// TwinCAT 3 PLC project plc_tmo_granite3_test
// ProgramVersion: 3.1.4022.7
// libraries:
//   LCLS General, * (SLAC)
//   lcls-twincat-motion, * (SLAC)
//   lcls2-cc-lib, * (SLAC)
//   PMPS, * (SLAC - LCLS)
//   Tc2_Standard, * (Beckhoff Automation GmbH)
//   Tc2_System, * (Beckhoff Automation GmbH)
//   Tc3_Module, * (Beckhoff Automation GmbH)
//   Tc2_MC2,3.3.42.0,Beckhoff Automation GmbH
// project tree:
//   DUTs/ E_HomeState.TcDUT (not stored)
//   GVLs/ GVL_PMPS.TcGVL (not stored), Main.TcGVL
//   / PlcTask.TcTTO
//   POUs/ PRG_1_PlcTask.TcPOU (not stored), PRG_2_PMPS_PRE.TcPOU (not stored), PRG_3_PMPS_POST.TcPOU (not stored), PRG_4_LOG.TcPOU (not stored), PRG_AL1K4_L2SI.TcPOU (not stored), PRG_IM2K4_PPM.TcPOU (not stored), PRG_IM3K4_PPM.TcPOU (not stored), PRG_IM4K4_PPM.TcPOU (not stored), PRG_IM5K4_PPM.TcPOU (not stored), PRG_IM6K4_PPM.TcPOU (not stored), PRG_LI1K4_IP1.TcPOU (not stored), PRG_PF1K4_WFS_TARGET.TcPOU (not stored), PRG_PF2K4_WFS_TARGET.TcPOU, PRG_SL1K4_SCATTER.TcPOU (not stored), PRG_SL2K4_SCATTER.TcPOU (not stored), PRG_ST4K4_TMO_TERM.TcPOU (not stored), PRG_ST5K4_TMO_TERM_FIXED.TcPOU, PRG_TM1K4.TcPOU, PRG_TM2K4.TcPOU
//   POUs/temp/ FB_SLITS.TcPOU (not stored), FB_SLITS_POWER.TcPOU (not stored), FB_SLITS_SCATTER.TcPOU (not stored)
//   POUs/TM1K4/ ENUM_TM1K4_States.TcDUT (not stored), FB_TM1K4.TcPOU (not stored), FB_TM1K4_States.TcPOU (not stored)
// real-time tasks:
//   TASK PlcTask: cycle T#10ms, priority 20, ADS port 350
// motion (NC):
//   TASK NC-Task 1 SAF: cycle T#2ms, priority 4, ADS port 501
//   TASK NC-Task 1 SVB: cycle T#10ms, priority 8, ADS port 511
//   AXIS Axis 1 AL1K4-L2SI-MMS (id 1)
//     Dynamic: AccelerationMaximum=200, DecelerationMaximum=200, Acceleration=200, Deceleration=200, Jerk=500, DelayTime=0.004
//     Velo: Maximum=10
//     TargetPosControl: Range=0.002, Time=2
//     OtherSettings: AllowMotionCmdToSlave=true
//     encoder EncType=29
//       EncPara: ScaleFactorNumerator=5e-05, Offset=-214686.941, MaxCount=#xffffffff, ReferenceSystem=1
//         SoftEndMinControl: Enable=true, Range=-108.74
//         SoftEndMaxControl: Enable=true, Range=-33.49
//         Inc: RefSoftSyncMask=#x0000ffff
//     drive DrvType=24
//       Analog: VeloReferenz=100, ScaleFactorActTorque=0.1
//       TimeComp: TaskDelayCycles=1
//     controller CtrType=2
//       CtrPara: PriorControlFactor=1
//         PosDiffControl: Range=1
//         PID: PosKp=20, PosExtKp=1, PosExtVelo=0.1, DeadBandPosition=0.002
//         Observer: BandWidth=20
//   AXIS Axis 2 (id 2)
//     OtherSettings: AllowMotionCmdToSlave=true
//     encoder EncType=1
//     drive DrvType=5
//       Analog: ScaleFactorActTorque=0.1
//       TimeComp: TaskDelayCycles=1
//     controller CtrType=1
//       CtrPara: PriorControlFactor=1
//         Observer: BandWidth=20
//   AXIS Axis 3 (id 3)
//     OtherSettings: AllowMotionCmdToSlave=true
//     encoder EncType=1
//     drive DrvType=5
//       Analog: ScaleFactorActTorque=0.1
//       TimeComp: TaskDelayCycles=1
//     controller CtrType=1
//       CtrPara: PriorControlFactor=1
//         Observer: BandWidth=20
//   AXIS Axis 4 (id 4)
//     OtherSettings: AllowMotionCmdToSlave=true
//     encoder EncType=1
//     drive DrvType=5
//       Analog: ScaleFactorActTorque=0.1
//       TimeComp: TaskDelayCycles=1
//     controller CtrType=1
//       CtrPara: PriorControlFactor=1
//         Observer: BandWidth=20
//   AXIS Axis 5 (id 5)
//     OtherSettings: AllowMotionCmdToSlave=true
//     encoder EncType=1
//     drive DrvType=5
//       Analog: ScaleFactorActTorque=0.1
//       TimeComp: TaskDelayCycles=1
//     controller CtrType=1
//       CtrPara: PriorControlFactor=1
//         Observer: BandWidth=20
//   AXIS Axis 6 IM1K4-XTES-MMS (id 6)
//     Velo: Maximum=10
//     OtherSettings: AllowMotionCmdToSlave=true
//     encoder EncType=29
//       EncPara: ScaleFactorNumerator=5e-05, Offset=-398.1892, MaxCount=#x00400000, ReferenceSystem=1
//         SoftEndMinControl: Enable=true, Range=-90
//         SoftEndMaxControl: Enable=true
//         Inc: RefSoftSyncMask=#x00000000
//     drive DrvType=24
//       DrvPara: Inverse=true
//         Analog: VeloReferenz=50, ScaleFactorActTorque=0.1
//         TimeComp: TaskDelayCycles=1
//     controller CtrType=2
//       CtrPara: PriorControlFactor=1
//         PosDiffControl: Range=1
//         PID: PosKp=20, PosExtKp=20, DeadBandPosition=0.001
//         Observer: BandWidth=20
//   AXIS Axis 7 IM1K4-XTES-CLZ (id 7)
//     General: UnitName=%
//     Velo: Maximum=10
//     OtherSettings: AllowMotionCmdToSlave=true
//     encoder EncType=4
//       EncPara: ScaleFactorNumerator=0.003, MaxCount=#x0000ffff
//         SoftEndMinControl: Enable=true, Range=-100
//         SoftEndMaxControl: Enable=true, Range=100
//         Inc: RefSoftSyncMask=#x0000ffff
//     drive DrvType=23
//       DrvPara: Inverse=true
//         Analog: VeloReferenz=33, ScaleFactorActTorque=0.1
//         TimeComp: TaskDelayCycles=1
//     controller CtrType=2
//       CtrPara: PriorControlFactor=1
//         PosDiffControl: Range=1
//         PID: PosKp=20, PosExtKp=20, DeadBandPosition=0.1
//         Observer: BandWidth=20
//   AXIS Axis 8 IM1K4-XTES-CLF (id 8)
//     General: UnitName=%
//     Velo: Maximum=10
//     OtherSettings: AllowMotionCmdToSlave=true
//     encoder EncType=4
//       EncPara: ScaleFactorNumerator=0.008, MaxCount=#x0000ffff
//         SoftEndMinControl: Enable=true, Range=-100
//         SoftEndMaxControl: Enable=true, Range=100
//         Inc: RefSoftSyncMask=#x0000ffff
//     drive DrvType=23
//       DrvPara: Inverse=true
//         Analog: VeloReferenz=70, ScaleFactorActTorque=0.1
//         TimeComp: TaskDelayCycles=1
//     controller CtrType=2
//       CtrPara: PriorControlFactor=1
//         PosDiffControl: Range=1
//         PID: PosKp=20, PosExtKp=20, DeadBandPosition=0.1
//         Observer: BandWidth=20
//   AXIS Axis 9 IM2K4-PPM-MMS (id 9)
//     Dynamic: AccelerationMaximum=200, DecelerationMaximum=200, Acceleration=200, Deceleration=200, Jerk=500, DelayTime=0.004
//     Velo: Maximum=65
//     TargetPosControl: Range=0.002, Time=2
//     OtherSettings: AllowMotionCmdToSlave=true
//     encoder EncType=29
//       EncPara: ScaleFactorNumerator=5e-05, Offset=-358.0066, MaxCount=#x00400000, ReferenceSystem=1
//         SoftEndMinControl: Enable=true, Range=-100.57
//         SoftEndMaxControl: Enable=true, Range=-7.67
//         Inc: RefSoftSyncMask=#x00000000
//     drive DrvType=24
//       Analog: VeloReferenz=100, ScaleFactorActTorque=0.1
//       TimeComp: TaskDelayCycles=1
//     controller CtrType=2
//       CtrPara: PriorControlFactor=1
//         PosDiffControl: Range=1
//         PID: PosKp=20, PosExtKp=1, PosExtVelo=0.1, DeadBandPosition=0.002
//         Observer: BandWidth=20
//   AXIS SL1K4-BOTTOM-M10 (id 10)
//     Velo: Maximum=2.2
//     OtherSettings: AllowMotionCmdToSlave=true
//     encoder EncType=4
//       EncPara: MaxCount=#x0000ffff
//         SoftEndMinControl: Enable=true, Range=-31.51
//         SoftEndMaxControl: Enable=true
//         Inc: RefSoftSyncMask=#x0000ffff
//     drive DrvType=24
//       Analog: VeloReferenz=2, ScaleFactorActTorque=0.1
//       TimeComp: TaskDelayCycles=1
//     controller CtrType=1
//       CtrPara: PriorControlFactor=1
//         PosDiffControl: Range=0.05
//         Observer: BandWidth=20
//   AXIS SL1K4-TOP-M11 (id 11)
//     Velo: Maximum=2.2
//     OtherSettings: AllowMotionCmdToSlave=true
//     encoder EncType=4
//       EncPara: Inverse=true, MaxCount=#x0000ffff
//         SoftEndMinControl: Enable=true, Range=-31.99
//         SoftEndMaxControl: Enable=true
//         Inc: RefSoftSyncMask=#x0000ffff
//     drive DrvType=24
//       Analog: VeloReferenz=2, ScaleFactorActTorque=0.1
//       TimeComp: TaskDelayCycles=1
//     controller CtrType=1
//       CtrPara: PriorControlFactor=1
//         PosDiffControl: Range=0.05
//         Observer: BandWidth=20
//   AXIS SL1K4-NORTH-M12 (id 12)
//     Velo: Maximum=2.2
//     OtherSettings: AllowMotionCmdToSlave=true
//     encoder EncType=4
//       EncPara: Inverse=true, MaxCount=#x0000ffff
//         SoftEndMinControl: Enable=true, Range=-31.5
//         SoftEndMaxControl: Enable=true
//         Inc: RefSoftSyncMask=#x0000ffff
//     drive DrvType=24
//       Analog: VeloReferenz=2, ScaleFactorActTorque=0.1
//       TimeComp: TaskDelayCycles=1
//     controller CtrType=1
//       CtrPara: PriorControlFactor=1
//         PosDiffControl: Range=0.05
//         Observer: BandWidth=20
//   AXIS SL1K4-SOUTH-M13 (id 13)
//     Velo: Maximum=2.2
//     OtherSettings: AllowMotionCmdToSlave=true
//     encoder EncType=4
//       EncPara: MaxCount=#x0000ffff
//         SoftEndMinControl: Enable=true, Range=-30.29
//         SoftEndMaxControl: Enable=true
//         Inc: RefSoftSyncMask=#x0000ffff
//     drive DrvType=24
//       Analog: VeloReferenz=2, ScaleFactorActTorque=0.1
//       TimeComp: TaskDelayCycles=1
//     controller CtrType=1
//       CtrPara: PriorControlFactor=1
//         PosDiffControl: Range=0.05
//         Observer: BandWidth=20
//   AXIS ST1K4-TEST (id 14)
//     Velo: RefSearch=5, RefSync=5, SlowManual=1, FastManual=5, Maximum=50
//     OtherSettings: AllowMotionCmdToSlave=true
//     encoder EncType=4
//       EncPara: ScaleFactorNumerator=0.000390625, Inverse=true, MaxCount=#x0000ffff
//         Inc: RefSoftSyncMask=#x0000ffff
//     drive DrvType=24
//       DrvPara: Inverse=true
//         Analog: VeloReferenz=50
//         TimeComp: TaskDelayCycles=1
//     controller CtrType=1
//       CtrPara: PriorControlFactor=1
//         PosDiffControl: Enable=false, Range=0.05
//         Observer: BandWidth=20
//   AXIS Axis 15 IM3K4-PPM-MMS (id 15)
//     Dynamic: AccelerationMaximum=200, DecelerationMaximum=200, Acceleration=200, Deceleration=200, Jerk=1000, DelayTime=0.004
//     Velo: Maximum=65
//     MotionControl: Enable=true, Range=0.0005, Time=1
//     TargetPosControl: Range=0.01, Time=1
//     OtherSettings: AllowMotionCmdToSlave=true
//     encoder EncType=29
//       EncPara: ScaleFactorNumerator=5e-05, Offset=-358.0066, MaxCount=#x00400000, ReferenceSystem=1
//         SoftEndMinControl: Enable=true, Range=-97.98
//         SoftEndMaxControl: Enable=true, Range=-5.69
//     drive DrvType=24
//       Analog: VeloReferenz=100, ScaleFactorActTorque=0.1
//       TimeComp: TaskDelayCycles=1
//     controller CtrType=2
//       CtrPara: PriorControlFactor=1
//         PosDiffControl: Range=10, Time=0.1
//         PID: PosKp=10, PosExtKp=0.01, PosExtVelo=0.0005, DeadBandPosition=0.0001
//         Observer: BandWidth=20
//   AXIS Axis 16 IM4K4-PPM-MMS (id 16)
//     Dynamic: AccelerationMaximum=200, DecelerationMaximum=200, Acceleration=200, Deceleration=200, Jerk=1000, DelayTime=0.004
//     Velo: Maximum=65
//     MotionControl: Enable=true, Range=0.0005, Time=1
//     TargetPosControl: Range=0.01, Time=1
//     OtherSettings: AllowMotionCmdToSlave=true
//     encoder EncType=29
//       EncPara: ScaleFactorNumerator=5e-05, Offset=-358.0066, MaxCount=#x00400000, ReferenceSystem=1
//         SoftEndMinControl: Enable=true, Range=-99.53
//         SoftEndMaxControl: Enable=true, Range=-8.43
//     drive DrvType=24
//       Analog: VeloReferenz=100, ScaleFactorActTorque=0.1
//       TimeComp: TaskDelayCycles=1
//     controller CtrType=2
//       CtrPara: PriorControlFactor=1
//         PosDiffControl: Range=10, Time=0.1
//         PID: PosKp=10, PosExtKp=0.01, PosExtVelo=0.0005, DeadBandPosition=0.0001
//         Observer: BandWidth=20
//   AXIS Axis 17 IM5K4-PPM-MMS (id 17)
//     Dynamic: AccelerationMaximum=200, DecelerationMaximum=200, Acceleration=200, Deceleration=200, Jerk=1000, DelayTime=0.004
//     Velo: Maximum=65
//     MotionControl: Enable=true, Range=0.0005, Time=1
//     TargetPosControl: Range=0.01, Time=1
//     OtherSettings: AllowMotionCmdToSlave=true
//     encoder EncType=29
//       EncPara: ScaleFactorNumerator=5e-05, Offset=-358.0066, MaxCount=#x00400000, ReferenceSystem=1
//         SoftEndMinControl: Enable=true, Range=-97.47
//         SoftEndMaxControl: Enable=true, Range=-4.42
//     drive DrvType=24
//       Analog: VeloReferenz=100, ScaleFactorActTorque=0.1
//       TimeComp: TaskDelayCycles=1
//     controller CtrType=2
//       CtrPara: PriorControlFactor=1
//         PosDiffControl: Range=10, Time=0.1
//         PID: PosKp=10, PosExtKp=0.01, PosExtVelo=0.0005, DeadBandPosition=0.0001
//         Observer: BandWidth=20
//   AXIS Axis 27 IM6K4-PPM-MMS (id 27)
//     Dynamic: AccelerationMaximum=200, DecelerationMaximum=200, Acceleration=200, Deceleration=200, Jerk=500, DelayTime=0.004
//     Velo: Maximum=65
//     TargetPosControl: Range=0.002, Time=2
//     OtherSettings: AllowMotionCmdToSlave=true
//     encoder EncType=29
//       EncPara: ScaleFactorNumerator=5e-05, Offset=-358.0066, MaxCount=#x00400000, ReferenceSystem=1
//         SoftEndMinControl: Enable=true, Range=-97.47
//         SoftEndMaxControl: Enable=true, Range=-4.42
//     drive DrvType=24
//       Analog: VeloReferenz=100, ScaleFactorActTorque=0.1
//       TimeComp: TaskDelayCycles=1
//     controller CtrType=2
//       CtrPara: PriorControlFactor=1
//         PosDiffControl: Range=10, Time=0.1
//         PID: PosKp=10, PosExtKp=0.01, PosExtVelo=0.0005, DeadBandPosition=0.0001
//         Observer: BandWidth=20
//   AXIS Axis 18 PF1K4-WFS_TARGET-MMS-Y (id 18)
//     Dynamic: AccelerationMaximum=200, DecelerationMaximum=200, Acceleration=10, Deceleration=10, Jerk=500, DelayTime=0.004
//     Velo: Maximum=20
//     TargetPosControl: Range=0.002, Time=2
//     OtherSettings: AllowMotionCmdToSlave=true
//     encoder EncType=29
//       EncPara: ScaleFactorNumerator=5e-05, Offset=-358.0066, MaxCount=#x00400000, ReferenceSystem=1
//         SoftEndMinControl: Enable=true, Range=-99.33
//         SoftEndMaxControl: Enable=true, Range=-9.71
//     drive DrvType=24
//       Analog: VeloReferenz=100, ScaleFactorActTorque=0.1
//       TimeComp: TaskDelayCycles=1
//     controller CtrType=2
//       CtrPara: PriorControlFactor=1
//         PosDiffControl: Range=1
//         PID: PosKp=20, PosExtKp=1, PosExtVelo=0.1, DeadBandPosition=0.002
//         Observer: BandWidth=20
//   AXIS Axis 19 PF1K4-WFS_TARGET-MMS-Z (id 19)
//     Dynamic: AccelerationMaximum=200, DecelerationMaximum=200, Acceleration=10, Deceleration=50, Jerk=500
//     Velo: Maximum=5
//     OtherSettings: AllowMotionCmdToSlave=true
//     encoder EncType=29
//       EncPara: ScaleFactorNumerator=5e-05, MaxCount=#x00400000, ReferenceSystem=1
//         SoftEndMinControl: Enable=true, Range=6.5
//         SoftEndMaxControl: Enable=true, Range=56
//     drive DrvType=24
//       DrvPara: Inverse=true
//         Analog: VeloReferenz=15.875, ScaleFactorActTorque=0.1
//         TimeComp: TaskDelayCycles=1
//     controller CtrType=1
//       CtrPara: PriorControlFactor=1
//         PosDiffControl: Range=1
//         Observer: BandWidth=20
//   AXIS Axis 28 PF2K4-WFS_TARGET-MMS-Y (id 28)
//     Dynamic: AccelerationMaximum=200, DecelerationMaximum=200, Acceleration=10, Deceleration=10, Jerk=500, DelayTime=0.004
//     Velo: Maximum=20
//     TargetPosControl: Range=0.002, Time=2
//     OtherSettings: AllowMotionCmdToSlave=true
//     encoder EncType=29
//       EncPara: ScaleFactorNumerator=5e-05, Offset=-358.0066, MaxCount=#x00400000, ReferenceSystem=1
//         SoftEndMinControl: Enable=true, Range=-99.33
//         SoftEndMaxControl: Enable=true, Range=-9.71
//     drive DrvType=24
//       Analog: VeloReferenz=100, ScaleFactorActTorque=0.1
//       TimeComp: TaskDelayCycles=1
//     controller CtrType=2
//       CtrPara: PriorControlFactor=1
//         PosDiffControl: Range=1
//         PID: PosKp=20, PosExtKp=1, PosExtVelo=0.1, DeadBandPosition=0.002
//         Observer: BandWidth=20
//   AXIS Axis 29 PF2K4-WFS_TARGET-MMS-Z (id 29)
//     Dynamic: AccelerationMaximum=200, DecelerationMaximum=200, Acceleration=10, Deceleration=50, Jerk=500
//     Velo: Maximum=5
//     OtherSettings: AllowMotionCmdToSlave=true
//     encoder EncType=29
//       EncPara: ScaleFactorNumerator=5e-05, MaxCount=#x00400000, ReferenceSystem=1
//         SoftEndMinControl: Enable=true, Range=6.5
//         SoftEndMaxControl: Enable=true, Range=56
//     drive DrvType=24
//       DrvPara: Inverse=true
//         Analog: VeloReferenz=15.875, ScaleFactorActTorque=0.1
//         TimeComp: TaskDelayCycles=1
//     controller CtrType=1
//       CtrPara: PriorControlFactor=1
//         PosDiffControl: Range=1
//         Observer: BandWidth=20
//   AXIS Axis 20 LI1K4-IP1-MMS (id 20)
//     Dynamic: AccelerationMaximum=200, DecelerationMaximum=200, Acceleration=200, Deceleration=200, Jerk=500, DelayTime=0.004
//     Velo: Maximum=65
//     TargetPosControl: Range=0.002, Time=2
//     OtherSettings: AllowMotionCmdToSlave=true
//     encoder EncType=29
//       EncPara: ScaleFactorNumerator=5e-05, Offset=-358.0066, MaxCount=#x00400000, ReferenceSystem=1
//         SoftEndMinControl: Enable=true, Range=-107.43
//         SoftEndMaxControl: Enable=true, Range=1.35
//     drive DrvType=24
//       Analog: VeloReferenz=100, ScaleFactorActTorque=0.1
//       TimeComp: TaskDelayCycles=1
//     controller CtrType=2
//       CtrPara: PriorControlFactor=1
//         PosDiffControl: Range=1
//         PID: PosKp=20, PosExtKp=1, PosExtVelo=0.1, DeadBandPosition=0.002
//         Observer: BandWidth=20
//   AXIS Axis 21 TM1K4-MMS-Y (id 21)
//     Dynamic: AccelerationMaximum=200, DecelerationMaximum=200, Acceleration=10, Deceleration=10, Jerk=500, DelayTime=0.004
//     Velo: Maximum=20
//     TargetPosControl: Range=0.002, Time=2
//     OtherSettings: AllowMotionCmdToSlave=true
//     encoder EncType=29
//       EncPara: ScaleFactorNumerator=5e-05, Offset=-358.0066, MaxCount=#x00400000, ReferenceSystem=1
//         SoftEndMinControl: Enable=true, Range=-102.55
//         SoftEndMaxControl: Enable=true, Range=1.41
//     drive DrvType=24
//       Analog: VeloReferenz=100, ScaleFactorActTorque=0.1
//       TimeComp: TaskDelayCycles=1
//     controller CtrType=2
//       CtrPara: PriorControlFactor=1
//         PosDiffControl: Range=1
//         PID: PosKp=20, PosExtKp=1, PosExtVelo=0.1, DeadBandPosition=0.002
//         Observer: BandWidth=20
//   AXIS Axis 22 TM1K4-MMS-X (id 22)
//     Dynamic: AccelerationMaximum=200, DecelerationMaximum=200, Acceleration=10, Deceleration=50, Jerk=500
//     Velo: Maximum=5
//     OtherSettings: AllowMotionCmdToSlave=true
//     encoder EncType=29
//       EncPara: ScaleFactorNumerator=5e-05, MaxCount=#x00400000, ReferenceSystem=1
//         SoftEndMinControl: Enable=true, Range=8.1
//         SoftEndMaxControl: Enable=true, Range=12.5
//     drive DrvType=24
//       Analog: VeloReferenz=15.875, ScaleFactorActTorque=0.1
//       TimeComp: TaskDelayCycles=1
//     controller CtrType=1
//       CtrPara: PriorControlFactor=1
//         PosDiffControl: Range=0.2
//         Observer: BandWidth=20
//   AXIS Axis 30 TM2K4-MMS-Y (id 30)
//     Dynamic: AccelerationMaximum=200, DecelerationMaximum=200, Acceleration=10, Deceleration=10, Jerk=500, DelayTime=0.004
//     Velo: Maximum=20
//     TargetPosControl: Range=0.002, Time=2
//     OtherSettings: AllowMotionCmdToSlave=true
//     encoder EncType=29
//       EncPara: ScaleFactorNumerator=5e-05, Offset=-358.0066, MaxCount=#x00400000, ReferenceSystem=1
//         SoftEndMinControl: Enable=true, Range=-102.55
//         SoftEndMaxControl: Enable=true, Range=1.41
//     drive DrvType=24
//       Analog: VeloReferenz=100, ScaleFactorActTorque=0.1
//       TimeComp: TaskDelayCycles=1
//     controller CtrType=2
//       CtrPara: PriorControlFactor=1
//         PosDiffControl: Range=1
//         PID: PosKp=20, PosExtKp=1, PosExtVelo=0.1, DeadBandPosition=0.002
//         Observer: BandWidth=20
//   AXIS Axis 31 TM2K4-MMS-X (id 31)
//     Dynamic: AccelerationMaximum=200, DecelerationMaximum=200, Acceleration=10, Deceleration=50, Jerk=500
//     Velo: Maximum=5
//     OtherSettings: AllowMotionCmdToSlave=true
//     encoder EncType=29
//       EncPara: ScaleFactorNumerator=5e-05, MaxCount=#x00400000, ReferenceSystem=1
//         SoftEndMinControl: Enable=true, Range=8.1
//         SoftEndMaxControl: Enable=true, Range=12.5
//     drive DrvType=24
//       Analog: VeloReferenz=15.875, ScaleFactorActTorque=0.1
//       TimeComp: TaskDelayCycles=1
//     controller CtrType=1
//       CtrPara: PriorControlFactor=1
//         PosDiffControl: Range=0.2
//         Observer: BandWidth=20
//   AXIS SL2K4-BOTTOM-M23 (id 23) // C:\Github\lcls-plc-tmo-motion\plc-tmo-motion\_Config\NC\Axes\SL2K4-BOTTOM-M23.xti
//     Velo: RefSearch=0.2, RefSync=0.05, Maximum=2.2
//     OtherSettings: AllowMotionCmdToSlave=true
//     encoder EncType=4
//       EncPara: MaxCount=#x0000ffff
//         SoftEndMinControl: Enable=true, Range=-30.61
//         SoftEndMaxControl: Enable=true
//         Inc: RefSoftSyncMask=#x0000ffff
//     drive DrvType=24
//       Analog: VeloReferenz=2, ScaleFactorActTorque=0.1
//       TimeComp: TaskDelayCycles=1
//     controller CtrType=1
//       CtrPara: PriorControlFactor=1
//         Observer: BandWidth=20
//   AXIS SL2K4-NORTH-M25 (id 25) // C:\Github\lcls-plc-tmo-motion\plc-tmo-motion\_Config\NC\Axes\SL2K4-NORTH-M25.xti
//     Velo: RefSearch=0.2, RefSync=0.05, Maximum=2.2
//     OtherSettings: AllowMotionCmdToSlave=true
//     encoder EncType=4
//       EncPara: Inverse=true, MaxCount=#x0000ffff
//         SoftEndMinControl: Enable=true, Range=-30.81
//         SoftEndMaxControl: Enable=true
//         Inc: RefSoftSyncMask=#x0000ffff
//     drive DrvType=24
//       Analog: VeloReferenz=2, ScaleFactorActTorque=0.1
//       TimeComp: TaskDelayCycles=1
//     controller CtrType=1
//       CtrPara: PriorControlFactor=1
//         Observer: BandWidth=20
//   AXIS SL2K4-SOUTH-M26 (id 26) // C:\Github\lcls-plc-tmo-motion\plc-tmo-motion\_Config\NC\Axes\SL2K4-SOUTH-M26.xti
//     Velo: RefSearch=0.2, RefSync=0.05, Maximum=2.2
//     OtherSettings: AllowMotionCmdToSlave=true
//     encoder EncType=4
//       EncPara: MaxCount=#x0000ffff
//         SoftEndMinControl: Enable=true, Range=-30.52
//         SoftEndMaxControl: Enable=true
//         Inc: RefSoftSyncMask=#x0000ffff
//     drive DrvType=24
//       Analog: VeloReferenz=2, ScaleFactorActTorque=0.1
//       TimeComp: TaskDelayCycles=1
//     controller CtrType=1
//       CtrPara: PriorControlFactor=1
//         Observer: BandWidth=20
//   AXIS SL2K4-TOP-M24 (id 24) // C:\Github\lcls-plc-tmo-motion\plc-tmo-motion\_Config\NC\Axes\SL2K4-TOP-M24.xti
//     Velo: RefSearch=0.2, RefSync=0.05, Maximum=2.2
//     PositionAreaControl: Range=0.5
//     TargetPosControl: Range=0.1
//     OtherSettings: AllowMotionCmdToSlave=true
//     encoder EncType=4
//       EncPara: Inverse=true, MaxCount=#x0000ffff
//         SoftEndMinControl: Enable=true, Range=-30.91
//         SoftEndMaxControl: Enable=true
//         Inc: RefSoftSyncMask=#x0000ffff
//     drive DrvType=24
//       Analog: VeloReferenz=2, ScaleFactorActTorque=0.1
//       TimeComp: TaskDelayCycles=1
//     controller CtrType=1
//       CtrPara: PriorControlFactor=1
//         PosDiffControl: Range=0.5
//         Observer: BandWidth=20
// I/O:
//   DEVICE Device 1 (EtherCAT), AmsNetId 172.21.132.155.2.1
//     PLC_EK1200 [EK1200-5000 EtherCAT Power supply (2A E-Bus)]
//       Coupler_EK1110 [EK1110 EtherCAT extension]

CONFIGURATION plc_tmo_granite3_test
    RESOURCE PLC ON TwinCAT3
        TASK PlcTask(INTERVAL := T#10ms, PRIORITY := 20);
        PROGRAM PRG_1_PlcTask WITH PlcTask : PRG_1_PlcTask;
    END_RESOURCE
END_CONFIGURATION

// ---- GVLs/Main.TcGVL
{attribute 'qualified_only'}
VAR_GLOBAL
    // AL1K4-L2SI: 1 Axis
    {attribute 'pytmc' := 'pv: AL1K4:L2SI:MMS'}
    {attribute 'TcLinkTo' := '.bLimitForwardEnable  := TIIB[AL1K4-EL7041-E1]^STM Status^Status^Digital input 1;
                              .bLimitBackwardEnable := TIIB[AL1K4-EL7041-E1]^STM Status^Status^Digital input 2;
                              .bBrakeRelease        := TIIB[AL1K4-EL2004-E3]^Channel 1^Output;
                              .nRawEncoderULINT     := TIIB[AL1K4-EL5042-E2]^FB Inputs Channel 1^Position'}
    M1: DUT_MotionStage := (sName := 'AL1K4:L2SI:MMS');

    // SPARE: 7 Axes (formerly AT1K4-SOLID and IM1K4-XTES)
    M2: DUT_MotionStage;
    M3: DUT_MotionStage;
    M4: DUT_MotionStage;
    M5: DUT_MotionStage;
    M6: DUT_MotionStage;
    M7: DUT_MotionStage;
    M8: DUT_MotionStage;

    // IM2K4-PPM: 1 Axis
    {attribute 'pytmc' := 'pv: IM2K4:PPM:MMS'}
    {attribute 'TcLinkTo' := '.bLimitForwardEnable  := TIIB[IM2K4-EL7041-E1]^STM Status^Status^Digital input 1;
                              .bLimitBackwardEnable := TIIB[IM2K4-EL7041-E1]^STM Status^Status^Digital input 2;
                              .bBrakeRelease        := TIIB[IM2K4-EL2004-E3]^Channel 1^Output;
                              .nRawEncoderULINT     := TIIB[IM2K4-EL5042-E2]^FB Inputs Channel 1^Position'}
    M9: DUT_MotionStage := (sName := 'IM2K4:PPM:MMS');

    // SL1K4-SCATTER: 4 Axes
    {attribute 'pytmc' := 'pv: SL1K4:SCATTER:MMS:BOTTOM'}
    {attribute 'TcLinkTo' := '.bLimitForwardEnable  := TIIB[SL1K4-EL7031-E1]^STM Status^Status^Digital input 2;
                              .bLimitBackwardEnable := TIIB[SL1K4-EL7031-E1]^STM Status^Status^Digital input 1;
                              .nRawEncoderUINT      := TIIB[SL1K4-EL5101-E2]^ENC Status compact^Counter value'}
    M10: DUT_MotionStage := (sName := 'SL1K4:SCATTER:MMS:BOTTOM');
    {attribute 'pytmc' := 'pv: SL1K4:SCATTER:MMS:TOP'}
    {attribute 'TcLinkTo' := '.bLimitForwardEnable  := TIIB[SL1K4-EL7031-E3]^STM Status^Status^Digital input 2;
                              .bLimitBackwardEnable := TIIB[SL1K4-EL7031-E3]^STM Status^Status^Digital input 1;
                              .nRawEncoderUINT      := TIIB[SL1K4-EL5101-E4]^ENC Status compact^Counter value'}
    M11: DUT_MotionStage := (sName := 'SL1K4:SCATTER:MMS:TOP');
    {attribute 'pytmc' := 'pv: SL1K4:SCATTER:MMS:NORTH'}
    {attribute 'TcLinkTo' := '.bLimitForwardEnable  := TIIB[SL1K4-EL7031-E5]^STM Status^Status^Digital input 1;
                              .bLimitBackwardEnable := TIIB[SL1K4-EL7031-E5]^STM Status^Status^Digital input 2;
                              .nRawEncoderUINT      := TIIB[SL1K4-EL5101-E6]^ENC Status compact^Counter value'}
    M12: DUT_MotionStage := (sName := 'SL1K4:SCATTER:MMS:NORTH');
    {attribute 'pytmc' := 'pv: SL1K4:SCATTER:MMS:SOUTH'}
    {attribute 'TcLinkTo' := '.bLimitForwardEnable  := TIIB[SL1K4-EL7031-E7]^STM Status^Status^Digital input 1;
                              .bLimitBackwardEnable := TIIB[SL1K4-EL7031-E7]^STM Status^Status^Digital input 2;
                              .nRawEncoderUINT      := TIIB[SL1K4-EL5101-E8]^ENC Status compact^Counter value'}
    M13: DUT_MotionStage := (sName := 'SL1K4:SCATTER:MMS:SOUTH');

    // SPARE: 1 Axis (formerly ST1K4-TEST)
    M14: DUT_MotionStage;

    // IM3K4-PPM: 1 Axis
    {attribute 'pytmc' := 'pv: IM3K4:PPM:MMS'}
    {attribute 'TcLinkTo' := '.bLimitForwardEnable  := TIIB[IM3K4-EL7041-E1]^STM Status^Status^Digital input 1;
                              .bLimitBackwardEnable := TIIB[IM3K4-EL7041-E1]^STM Status^Status^Digital input 2;
                              .bBrakeRelease        := TIIB[IM3K4-EL2004-E3]^Channel 1^Output;
                              .nRawEncoderULINT     := TIIB[IM3K4-EL5042-E2]^FB Inputs Channel 1^Position'}
    M15: DUT_MotionStage := (sName := 'IM3K4:PPM:MMS');
    // IM4K4-PPM: 1 Axis
    {attribute 'pytmc' := 'pv: IM4K4:PPM:MMS'}
    {attribute 'TcLinkTo' := '.bLimitForwardEnable  := TIIB[IM4K4-EL7041-E1]^STM Status^Status^Digital input 1;
                              .bLimitBackwardEnable := TIIB[IM4K4-EL7041-E1]^STM Status^Status^Digital input 2;
                              .bBrakeRelease        := TIIB[IM4K4-EL2004-E3]^Channel 1^Output;
                              .nRawEncoderULINT     := TIIB[IM4K4-EL5042-E2]^FB Inputs Channel 1^Position'}
    M16: DUT_MotionStage := (sName := 'IM4K4:PPM:MMS');

    // IM5K4-PPM: 1 Axis
    {attribute 'pytmc' := 'pv: IM5K4:PPM:MMS'}
    {attribute 'TcLinkTo' := '.bLimitForwardEnable  := TIIB[IM5K4-EL7041-E1]^STM Status^Status^Digital input 1;
                              .bLimitBackwardEnable := TIIB[IM5K4-EL7041-E1]^STM Status^Status^Digital input 2;
                              .bBrakeRelease        := TIIB[IM5K4-EL2004-E3]^Channel 1^Output;
                              .nRawEncoderULINT     := TIIB[IM5K4-EL5042-E2]^FB Inputs Channel 1^Position'}
    M17: DUT_MotionStage := (sName := 'IM5K4:PPM:MMS');
	
    // PF1K4-WFS_TARGET: 2 Axes
    {attribute 'pytmc' := 'pv: PF1K4:WFS:MMS:Y'}
    {attribute 'TcLinkTo' := '.bLimitForwardEnable  := TIIB[PF1K4-EL7041-E1]^STM Status^Status^Digital input 1;
                              .bLimitBackwardEnable := TIIB[PF1K4-EL7041-E1]^STM Status^Status^Digital input 2;
                              .bBrakeRelease        := TIIB[PF1K4-EL2004-E4]^Channel 1^Output;
                              .nRawEncoderULINT     := TIIB[PF1K4-EL5042-E3]^FB Inputs Channel 2^Position'}
    M18: DUT_MotionStage := (sName := 'PF1K4:WFS:MMS:Y');
    {attribute 'pytmc' := 'pv: PF1K4:WFS:MMS:Z'}
    {attribute 'TcLinkTo' := '.nRawEncoderULINT     := TIIB[PF1K4-EL5042-E3]^FB Inputs Channel 1^Position'}
    M19: DUT_MotionStage := (sName := 'PF1K4:WFS:MMS:Z');
	
    // LI1K4-IP1: 1 Axis
    {attribute 'pytmc' := 'pv: LI1K4:IP1:MMS'}
    {attribute 'TcLinkTo' := '.bLimitForwardEnable  := TIIB[LI1K4-EL7041-E1]^STM Status^Status^Digital input 1;
                              .bLimitBackwardEnable := TIIB[LI1K4-EL7041-E1]^STM Status^Status^Digital input 2;
                              .bBrakeRelease        := TIIB[LI1K4-EL2004-E3]^Channel 1^Output;
                              .nRawEncoderULINT     := TIIB[LI1K4-EL5042-E2]^FB Inputs Channel 1^Position'}
    M20: DUT_MotionStage := (sName := 'LI1K4:IP1:MMS');

    // TM1K4: 2 Axes
    {attribute 'pytmc' := 'pv: TM1K4:ATM:MMS:Y'}
    {attribute 'TcLinkTo' := '.bLimitForwardEnable  := TIIB[TM1K4-EL7041-E1]^STM Status^Status^Digital input 1;
                              .bLimitBackwardEnable := TIIB[TM1K4-EL7041-E1]^STM Status^Status^Digital input 2;
                              .bBrakeRelease        := TIIB[TM1K4-EL2004-E4]^Channel 1^Output;
                              .nRawEncoderULINT     := TIIB[TM1K4-EL5042-E3]^FB Inputs Channel 1^Position'}
    M21: DUT_MotionStage := (sName := 'TM1K4:ATM:MMS:Y');
    {attribute 'pytmc' := 'pv: TM1K4:ATM:MMS:X'}
    {attribute 'TcLinkTo' := '.nRawEncoderULINT     := TIIB[TM1K4-EL5042-E3]^FB Inputs Channel 2^Position'}
    M22: DUT_MotionStage := (sName := 'TM1K4:ATM:MMS:X');

     // SL2K4-SCATTER: 4 Axes
    {attribute 'pytmc' := 'pv: SL2K4:SCATTER:MMS:BOTTOM'}
    {attribute 'TcLinkTo' := '.bLimitForwardEnable  := TIIB[SL2K4-EL7031-E1]^STM Status^Status^Digital input 2;
                             .bLimitBackwardEnable := TIIB[SL2K4-EL7031-E1]^STM Status^Status^Digital input 1;
                              .nRawEncoderUINT      := TIIB[SL2K4-EL5101-E2]^ENC Status compact^Counter value'}
    M23: DUT_MotionStage := (sName := 'SL2K4:SCATTER:MMS:BOTTOM');
    {attribute 'pytmc' := 'pv: SL2K4:SCATTER:MMS:TOP'}
    {attribute 'TcLinkTo' := '.bLimitForwardEnable  := TIIB[SL2K4-EL7031-E3]^STM Status^Status^Digital input 2;
                              .bLimitBackwardEnable := TIIB[SL2K4-EL7031-E3]^STM Status^Status^Digital input 1;
                              .nRawEncoderUINT      := TIIB[SL2K4-EL5101-E4]^ENC Status compact^Counter value'}
    M24: DUT_MotionStage := (sName := 'SL2K4:SCATTER:MMS:TOP');
    {attribute 'pytmc' := 'pv: SL2K4:SCATTER:MMS:NORTH'}
    {attribute 'TcLinkTo' := '.bLimitForwardEnable  := TIIB[SL2K4-EL7031-E5]^STM Status^Status^Digital input 1;
                              .bLimitBackwardEnable := TIIB[SL2K4-EL7031-E5]^STM Status^Status^Digital input 2;
                              .nRawEncoderUINT      := TIIB[SL2K4-EL5101-E6]^ENC Status compact^Counter value'}
    M25: DUT_MotionStage := (sName := 'SL2K4:SCATTER:MMS:NORTH');
    {attribute 'pytmc' := 'pv: SL2K4:SCATTER:MMS:SOUTH'}
    {attribute 'TcLinkTo' := '.bLimitForwardEnable  := TIIB[SL2K4-EL7031-E7]^STM Status^Status^Digital input 1;
                              .bLimitBackwardEnable := TIIB[SL2K4-EL7031-E7]^STM Status^Status^Digital input 2;
                              .nRawEncoderUINT      := TIIB[SL2K4-EL5101-E8]^ENC Status compact^Counter value'}
    M26: DUT_MotionStage := (sName := 'SL2K4:SCATTER:MMS:SOUTH');
	
	
// Granite 3 CCMs

    // IM6K4-PPM: 1 Axis
    {attribute 'pytmc' := 'pv: IM6K4:PPM:MMS'}
    {attribute 'TcLinkTo' := '.bLimitForwardEnable  := TIIB[IM6K4-EL7041-E1]^STM Status^Status^Digital input 1;
                              .bLimitBackwardEnable := TIIB[IM6K4-EL7041-E1]^STM Status^Status^Digital input 2;
                              .bBrakeRelease        := TIIB[IM6K4-EL2004-E3]^Channel 1^Output;
                              .nRawEncoderULINT     := TIIB[IM6K4-EL5042-E2]^FB Inputs Channel 1^Position'}
    M27: DUT_MotionStage := (sName := 'IM6K4:PPM:MMS');
	
	// PF2K4-WFS_TARGET: 2 Axes
	{attribute 'pytmc' := 'pv: PF2K4:WFS:MMS:Y'}
    {attribute 'TcLinkTo' := '.bLimitForwardEnable  := TIIB[PF2K4-EL7041-E1]^STM Status^Status^Digital input 1;
                              .bLimitBackwardEnable := TIIB[PF2K4-EL7041-E1]^STM Status^Status^Digital input 2;
                              .bBrakeRelease        := TIIB[PF2K4-EL2004-E4]^Channel 1^Output;
                              .nRawEncoderULINT     := TIIB[PF2K4-EL5042-E3]^FB Inputs Channel 2^Position'}
    M28: DUT_MotionStage := (sName := 'PF2K4:WFS:MMS:Y');
    {attribute 'pytmc' := 'pv: PF2K4:WFS:MMS:Z'}
    {attribute 'TcLinkTo' := '.nRawEncoderULINT     := TIIB[PF2K4-EL5042-E3]^FB Inputs Channel 1^Position'}
    M29: DUT_MotionStage := (sName := 'PF2K4:WFS:MMS:Z');
	
	// TM2K4 2 Axes
	{attribute 'pytmc' := 'pv: TM2K4:ATM:MMS:Y'}
    {attribute 'TcLinkTo' := '.bLimitForwardEnable  := TIIB[TM2K4-EL7041-E1]^STM Status^Status^Digital input 1;
                              .bLimitBackwardEnable := TIIB[TM2K4-EL7041-E1]^STM Status^Status^Digital input 2;
                              .bBrakeRelease        := TIIB[TM2K4-EL2004-E4]^Channel 1^Output;
                              .nRawEncoderULINT     := TIIB[TM2K4-EL5042-E3]^FB Inputs Channel 1^Position'}
    M30: DUT_MotionStage := (sName := 'TM2K4:ATM:MMS:Y');
    {attribute 'pytmc' := 'pv: TM2K4:ATM:MMS:X'}
    {attribute 'TcLinkTo' := '.nRawEncoderULINT     := TIIB[TM2K4-EL5042-E3]^FB Inputs Channel 2^Position'}
    M31: DUT_MotionStage := (sName := 'TM2K4:ATM:MMS:X');
	
	
END_VAR

// ---- POUs/PRG_PF2K4_WFS_TARGET.TcPOU
PROGRAM PRG_PF2K4_WFS_TARGET
VAR
	{attribute 'pytmc' := '
        pv: PF2K4:WFS
        io: io
    '}
    {attribute 'TcLinkTo' := '.fbThermoCouple1.bError 		:= TIIB[PF2K4-EL3314-E5]^TC Inputs Channel 1^Status^Error;
                              .fbThermoCouple1.bUnderrange	:= TIIB[PF2K4-EL3314-E5]^TC Inputs Channel 1^Status^Underrange;
                              .fbThermoCouple1.bOverrange 	:= TIIB[PF2K4-EL3314-E5]^TC Inputs Channel 1^Status^Overrange;
                              .fbThermoCouple1.iRaw 		:= TIIB[PF2K4-EL3314-E5]^TC Inputs Channel 1^Value;
                              .fbThermoCouple2.bError 		:= TIIB[PF2K4-EL3314-E5]^TC Inputs Channel 2^Status^Error;
                              .fbThermoCouple2.bUnderrange 	:= TIIB[PF2K4-EL3314-E5]^TC Inputs Channel 2^Status^Underrange;
                              .fbThermoCouple2.bOverrange 	:= TIIB[PF2K4-EL3314-E5]^TC Inputs Channel 2^Status^Overrange;
                              .fbThermoCouple2.iRaw 		:= TIIB[PF2K4-EL3314-E5]^TC Inputs Channel 2^Value'}
    fbPF2K4: FB_WFS;

    stSiBP: ST_BeamParams := PMPS_GVL.cstFullBeam;
END_VAR

// Exclusion range specified by M. Seaberg 2021-5-19
stSiBP.neVRange := F_eVExcludeRange(1.75E3, 3.15E3);
// Drop transmission to 20%
stSiBP.nTran := 0.20;

fbPF2K4.nTransitionAssertionID := 16#3140;
fbPF2K4.nUnknownAssertionID := 16#3149;

fbPF2K4.stOut.fPosition := -10.5;
fbPF2K4.stOut.bUseRawCounts := FALSE;
fbPF2K4.stOut.nRequestAssertionID := 16#3141;
fbPF2K4.stOut.stBeamParams := PMPS_GVL.cstFullBeam;
fbPF2K4.stOut.bValid := TRUE;

fbPF2K4.stTarget1.fPosition := -93.033;
fbPF2K4.stTarget1.bUseRawCounts := FALSE;
fbPF2K4.stTarget1.nRequestAssertionID := 16#3142;
fbPF2K4.stTarget1.stBeamParams := stSiBP;
fbPF2K4.stTarget1.bValid := TRUE;

fbPF2K4.stTarget2.fPosition := -78.658;
fbPF2K4.stTarget2.bUseRawCounts := FALSE;
fbPF2K4.stTarget2.nRequestAssertionID := 16#3143;
fbPF2K4.stTarget2.stBeamParams := stSiBP;
fbPF2K4.stTarget2.bValid := TRUE;

fbPF2K4.stTarget3.fPosition := -64.282;
fbPF2K4.stTarget3.bUseRawCounts := FALSE;
fbPF2K4.stTarget3.nRequestAssertionID := 16#3144;
fbPF2K4.stTarget3.stBeamParams := stSiBP;
fbPF2K4.stTarget3.bValid := TRUE;

fbPF2K4.stTarget4.fPosition := -49.907;
fbPF2K4.stTarget4.bUseRawCounts := FALSE;
fbPF2K4.stTarget4.nRequestAssertionID := 16#3145;
fbPF2K4.stTarget4.stBeamParams := stSiBP;
fbPF2K4.stTarget4.bValid := TRUE;

fbPF2K4.stTarget5.fPosition := -35.533;
fbPF2K4.stTarget5.bUseRawCounts := FALSE;
fbPF2K4.stTarget5.nRequestAssertionID := 16#3146;
fbPF2K4.stTarget5.stBeamParams := stSiBP;
fbPF2K4.stTarget5.bValid := TRUE;

fbPF2K4(
    fbArbiter := fbArbiter,
    fbFFHWO := fbFastFaultOutput2,
    stYStage := Main.M28,
    stZStage := Main.M29);

END_PROGRAM

// ---- POUs/PRG_ST5K4_TMO_TERM_FIXED.TcPOU
PROGRAM PRG_ST5K4_TMO_TERM_FIXED
VAR
    {attribute 'pytmc' := 'pv: ST5K4:TMO_TERM_FIXED'}
    {attribute 'TcLinkTo' := 	'.i_xInsertedLS	:=	TIIB[ST5K4-EP2338]^Channel 4^Input;
                                 .i_xRetractedLS:=	TIIB[ST5K4-EP2338]^Channel 3^Input;
                                 .q_xInsert_DO	:=	TIIB[ST5K4-EP2338]^Channel 9^Output
    '}
    ST5K4: FB_MotionPneumaticActuator;
    ibPMPS_OK : BOOL;
END_VAR

ST5K4(
    ibInsertOK:= TRUE,
    ibRetractOK:= TRUE,
    ibPMPS_OK:= ibPMPS_OK,
    ibSingleCntrl:= TRUE ,
    ibCntrlHold:= TRUE,
    ibOverrideInterlock:= ,
    i_xReset:= ,
    stPneumaticActuator=> ,
    xMPS_OK=>  ,
    io_fbFFHWO:= fbFastFaultOutput2  ); // Do Stoppers send MPS FAULT?

END_PROGRAM

// ---- POUs/PRG_TM1K4.TcPOU
PROGRAM PRG_TM1K4
VAR
    {attribute 'pytmc' := '
        pv: TM1K4:ATM
        io: io
    '}
    {attribute 'TcLinkTo' := '.fbThermoCouple1.bError := TIIB[TM1K4-EL3314-E5]^TC Inputs Channel 1^Status^Error;
                              .fbThermoCouple1.bUnderrange := TIIB[TM1K4-EL3314-E5]^TC Inputs Channel 1^Status^Underrange;
                              .fbThermoCouple1.bOverrange := TIIB[TM1K4-EL3314-E5]^TC Inputs Channel 1^Status^Overrange;
                              .fbThermoCouple1.iRaw := TIIB[TM1K4-EL3314-E5]^TC Inputs Channel 1^Value'}
    fbTM1K4: FB_TM1K4;
END_VAR

fbTM1K4.nTransitionAssertionID := 16#5140;
fbTM1K4.nUnknownAssertionID := 16#5149;

fbTM1K4.stOut.fPosition := -2.558;
fbTM1K4.stOut.bUseRawCounts := FALSE;
fbTM1K4.stOut.nRequestAssertionID := 16#5141;
fbTM1K4.stOut.stBeamParams := PMPS_GVL.cstFullBeam;
fbTM1K4.stOut.bValid := TRUE;

fbTM1K4.stTarget1a.fPosition := -16.311;
fbTM1K4.stTarget1a.bUseRawCounts := FALSE;
fbTM1K4.stTarget1a.nRequestAssertionID := 16#5142;
fbTM1K4.stTarget1a.stBeamParams := PMPS_GVL.cstFullBeam;
fbTM1K4.stTarget1a.bValid := TRUE;

fbTM1K4.stTarget1b.fPosition := -25.282;
fbTM1K4.stTarget1b.bUseRawCounts := FALSE;
fbTM1K4.stTarget1b.nRequestAssertionID := 16#5143;
fbTM1K4.stTarget1b.stBeamParams := PMPS_GVL.cstFullBeam;
fbTM1K4.stTarget1b.bValid := TRUE;

fbTM1K4.stTarget2b.fPosition := -41.249;
fbTM1K4.stTarget2b.bUseRawCounts := FALSE;
fbTM1K4.stTarget2b.nRequestAssertionID := 16#5144;
fbTM1K4.stTarget2b.stBeamParams := PMPS_GVL.cstFullBeam;
fbTM1K4.stTarget2b.bValid := TRUE;

fbTM1K4.stTarget3a.fPosition := -55.414;
fbTM1K4.stTarget3a.bUseRawCounts := FALSE;
fbTM1K4.stTarget3a.nRequestAssertionID := 16#5145;
fbTM1K4.stTarget3a.stBeamParams := PMPS_GVL.cstFullBeam;
fbTM1K4.stTarget3a.bValid := TRUE;

fbTM1K4.stTarget3b.fPosition := -62.895;
fbTM1K4.stTarget3b.bUseRawCounts := FALSE;
fbTM1K4.stTarget3b.nRequestAssertionID := 16#5146;
fbTM1K4.stTarget3b.stBeamParams := PMPS_GVL.cstFullBeam;
fbTM1K4.stTarget3b.bValid := TRUE;

fbTM1K4.stTarget4.fPosition := -82.25;
fbTM1K4.stTarget4.bUseRawCounts := FALSE;
fbTM1K4.stTarget4.nRequestAssertionID := 16#5147;
fbTM1K4.stTarget4.stBeamParams := PMPS_GVL.cstFullBeam;
fbTM1K4.stTarget4.bValid := TRUE;

fbTM1K4.stTarget5.fPosition := -102.258;
fbTM1K4.stTarget5.bUseRawCounts := FALSE;
fbTM1K4.stTarget5.nRequestAssertionID := 16#5148;
fbTM1K4.stTarget5.stBeamParams := PMPS_GVL.cstFullBeam;
fbTM1K4.stTarget5.bValid := TRUE;

fbTM1K4(
    fbArbiter := fbArbiter,
    fbFFHWO := fbFastFaultOutput1,
    stYStage := Main.M21,
    stXStage := Main.M22);

END_PROGRAM

// ---- POUs/PRG_TM2K4.TcPOU
PROGRAM PRG_TM2K4
VAR
	{attribute 'pytmc' := '
        pv: TM2K4:ATM
        io: io
    '}
    {attribute 'TcLinkTo' := '.fbThermoCouple1.bError := TIIB[TM2K4-EL3314-E5]^TC Inputs Channel 1^Status^Error;
                              .fbThermoCouple1.bUnderrange := TIIB[TM2K4-EL3314-E5]^TC Inputs Channel 1^Status^Underrange;
                              .fbThermoCouple1.bOverrange := TIIB[TM2K4-EL3314-E5]^TC Inputs Channel 1^Status^Overrange;
                              .fbThermoCouple1.iRaw := TIIB[TM2K4-EL3314-E5]^TC Inputs Channel 1^Value'}
    fbTM2K4: FB_ATM;
END_VAR

fbTM2K4.nTransitionAssertionID := 16#5240;
fbTM2K4.nUnknownAssertionID := 16#5149;

fbTM2K4.stOut.fPosition := -15;
fbTM2K4.stOut.bUseRawCounts := FALSE;
fbTM2K4.stOut.nRequestAssertionID := 16#5241;
fbTM2K4.stOut.stBeamParams := PMPS_GVL.cstFullBeam;
fbTM2K4.stOut.bValid := TRUE;

fbTM2K4.stTarget1.fPosition := -39.124;
fbTM2K4.stTarget1.bUseRawCounts := FALSE;
fbTM2K4.stTarget1.nRequestAssertionID := 16#5242;
fbTM2K4.stTarget1.stBeamParams := PMPS_GVL.cstFullBeam;
fbTM2K4.stTarget1.bValid := TRUE;

fbTM2K4.stTarget2.fPosition := -53.5;
fbTM2K4.stTarget2.bUseRawCounts := FALSE;
fbTM2K4.stTarget2.nRequestAssertionID := 16#5243;
fbTM2K4.stTarget2.stBeamParams := PMPS_GVL.cstFullBeam;
fbTM2K4.stTarget2.bValid := TRUE;

fbTM2K4.stTarget3.fPosition := -67.874;
fbTM2K4.stTarget3.bUseRawCounts := FALSE;
fbTM2K4.stTarget3.nRequestAssertionID := 16#5244;
fbTM2K4.stTarget3.stBeamParams := PMPS_GVL.cstFullBeam;
fbTM2K4.stTarget3.bValid := TRUE;

fbTM2K4.stTarget4.fPosition := -82.25;
fbTM2K4.stTarget4.bUseRawCounts := FALSE;
fbTM2K4.stTarget4.nRequestAssertionID := 16#5245;
fbTM2K4.stTarget4.stBeamParams := PMPS_GVL.cstFullBeam;
fbTM2K4.stTarget4.bValid := TRUE;

fbTM2K4.stTarget5.fPosition := -96.623;
fbTM2K4.stTarget5.bUseRawCounts := FALSE;
fbTM2K4.stTarget5.nRequestAssertionID := 16#5246;
fbTM2K4.stTarget5.stBeamParams := PMPS_GVL.cstFullBeam;
fbTM2K4.stTarget5.bValid := TRUE;

fbTM2K4(
    fbArbiter := fbArbiter,
    fbFFHWO := fbFastFaultOutput1,
    stYStage := Main.M30,
    stXStage := Main.M31);

END_PROGRAM
